TYPE (* a Struct holding 2x1 Object IDs *)
  (* Version 1.0, 2026-05-28, Franz Höpfinger, Demmler Andreas Fahrzeugbau *)
  PACKAGE isobus::UT::Q::types;
  IMPORT eclipse4diac::core::TypeHash;
  IMPORT isobus::UT::Q::const::IDs::ID_NULL;
  s2x1ObjectIDs : STRUCT
    up : isobus::UT::Q::types::s1ObjectID := (u16ObjId := ID_NULL); (* forward, up, right, clockwise *)
    down : isobus::UT::Q::types::s1ObjectID := (u16ObjId := ID_NULL); (* backward, down, left, counter-clockwise *)
  END_STRUCT;
END_TYPE
